{attribute 'GeneratedUsingTerminal: EL3443-0000-0016'}
{attribute addProperty BoxType "EL3443-0000-0016"}
{attribute addProperty Id "Voltage_Last_Zero_CrossingAT %I*ULINT8"}
{attribute addProperty CRC "3439292703"}
{attribute addProperty Size "8"}
TYPE L3_Timing_CCFF711F EXTENDS InputBase_8311D824 :
STRUCT
	{attribute addProperty Name "Voltage_Last_Zero_Crossing"}
	Voltage_Last_Zero_Crossing AT %I* : ULINT;
END_STRUCT
END_TYPE

(* stored: Version 1.2.0.0, ProductVersion 3.1.4024.11
   DUT L3_Timing_CCFF711F: Id {c825eab2-49ff-424d-b858-93b77f23ce44} *)
